{attribute addProperty BoxType "EK1122-0000-0018"}
{attribute addProperty Id "Beckhoff_EL68xxsub_EK1100EK1100_179A0949162"}
{attribute addProperty CRC "2201812640"}
{attribute addProperty SizeInBites "16"}
{attribute addProperty SizeInBytes "2"}
TYPE Beckhoff_EL68xxEK1122_833CFEA0 EXTENDS EK1122_179A0949 :
STRUCT
	{attribute addProperty Name "Beckhoff_EL68xxsub_EK1100"}
	Beckhoff_EL68xxsub_EK1100 : EK1100_179A0949;
END_STRUCT
END_TYPE

(* stored: Version 1.2.0.0, ProductVersion 3.1.4024.9
   DUT Beckhoff_EL68xxEK1122_833CFEA0: Id {16ff8ff1-714c-4779-a6b7-bb819e71b5a5} *)
